INTERFACE PUBLIC I_TripResettable EXTENDS __System.IQueryInterface

METHOD TripReset : BOOL
END_METHOD

END_INTERFACE

(* stored: Version 1.1.0.1, ProductVersion 3.1.4024.12
   Itf I_TripResettable: Id {40411f41-26e3-420f-958e-fe6a2434408d}
   Method TripReset: Id {68858e7f-b233-4544-a010-c8ff6d14d1ba} *)
